// TIA Portal V16 export
// export: Created 2021-11-21T21:05:54.6301485Z, ExportSetting WithDefaults, WithReadOnly, DisplayName Totally Integrated Automation Portal, DisplayVersion V16 Update 3, DisplayName TIA Portal Version Control Interface, DisplayVersion V16 Update 2, DisplayName TIA Portal Openness, DisplayVersion V16 Update 3, DisplayName SINAMICS Startdrive Advanced, DisplayVersion V16, DisplayName SINAMICS Startdrive G130, G150, S120, S150, SINAMICS MV, S210, DisplayVersion V16, DisplayName SINAMICS Startdrive G110M, G120, G120C, G120D, G120P, DisplayVersion V16, DisplayName STEP 7 Professional, DisplayVersion V16 Update 3, DisplayName SIMATIC Energy Suite, DisplayVersion V16, DisplayName STEP 7 Safety, DisplayVersion V16, DisplayName WinCC Advanced, DisplayVersion V16 Update 3
VAR_GLOBAL   // PLC tag table "Tabella delle variabili standard"
   Clock_Byte AT %MB0 : Byte;
   Clock_10Hz AT %M0.0 : Bool;
   Clock_5Hz AT %M0.1 : Bool;
   "Clock_2.5Hz" AT %M0.2 : Bool;
   Clock_2Hz AT %M0.3 : Bool;
   "Clock_1.25Hz" AT %M0.4 : Bool;
   Clock_1Hz AT %M0.5 : Bool;
   "Clock_0.625Hz" AT %M0.6 : Bool;
   "Clock_0.5Hz" AT %M0.7 : Bool;
   System_Byte AT %MB1 : Byte;
   FirstScan AT %M1.0 : Bool;
   DiagStatusUpdate AT %M1.1 : Bool;
   AlwaysTRUE AT %M1.2 : Bool;
   AlwaysFALSE AT %M1.3 : Bool;
   Tag_1 AT %M5.0 : Bool;
   Tag_2 AT %M4.0 : Bool;
   Tag_3 AT %M5.1 : Bool;
   Tag_4 AT %M5.2 : Bool;
   Tag_5 AT %M5.3 : Bool;
   Tag_6 AT %M5.4 : Bool;
   Tag_7 AT %M5.5 : Bool;
   Tag_8 AT %M4.2 : Bool;
   Tag_9 AT %M4.3 : Bool;
   Tag_10 AT %M4.4 : Bool;
   Tag_11 AT %M4.5 : Bool;
   Tag_12 AT %M4.1 : Bool;
   Tag_14 AT %MD5 : UDInt;
   start AT %MD30 : DWord;
   Tag_13 AT %M60.0 : Bool;
   Tag_15 AT %M20.0 : Bool;
   Tag_16 AT %M6.0 : Bool;
   Tag_17 AT %M6.1 : Bool;
   active AT %M90.0 : LWord;
   active_1 AT %M10.0 : LWord;
   Tag_21 AT %M15.0 : Bool;
   Tag_22 AT %MD40 : DWord;
   Liv_medio AT %MB8 : Byte;
   Liv_alto AT %MB9 : Byte;
   Tag_23 AT %M8.3 : Bool;
   "alto_0.1" AT %M9.1 : Bool;
   "medio_0.0" AT %M8.0 : Bool;
   Tag_26 AT %M9.3 : Bool;
   "medio_0.1" AT %M8.1 : Bool;
   "medio_0.2" AT %M8.2 : Bool;
   "alto_0.2" AT %M9.2 : Bool;
   "alto_0.0" AT %M9.0 : Bool;
   PROBLEMA_ALTO AT %M60.1 : Bool;
   PROBLEMA_MED AT %M60.3 : Bool;
   Tag_24 AT %M74.2 : Bool;
   Tag_25 AT %M75.3 : Bool;
   MEDIO_UGUALE AT %M33.3 : Bool;
   Tag_27 AT %M54.4 : Bool;
   ALTO_UGUALE AT %M54.5 : Bool;
   Errore AT %MB10 : Byte;
   "errore_0.0" AT %M10.0 : Bool;
   "errore_0.1" AT %M10.1 : Bool;
   "errore_0.2" AT %M10.2 : Bool;
   check_M AT %M18.0 : Bool;
   check_A AT %M18.1 : Bool;
END_VAR
